# EPICS substitutions: support/ip_use/2-9/iocBoot/iocIpTest/asynRecord.substitutions
file "$(ASYN)/db/asynRecord.db"
{
pattern
{P           R         PORT    ADDR    OMAX  IMAX}
{ipTest:     asyn_1   serial1    0     256  256}
{ipTest:     asyn_2   serial2    0     256  256}
{ipTest:     asyn_3   serial3    0     256  256}
{ipTest:     asyn_4   serial4    0     256  256}
}
